// TIA Portal V21 export
TYPE "motorStopCtx"
   STRUCT
      "step" : USInt;
      stepTime : LTime;
      alm : "motorAlm";
      almWord { S7_SetPoint := 'True'} : Word;
   END_STRUCT;
END_TYPE
